{attribute 'qualified_only'}
{attribute 'strict'}
{attribute 'to_string'}
TYPE EOpenDichtSchuifStatus :
(
	Open := 0,
	Dicht,
	Error,
	Openen,
	Sluiten
);
END_TYPE

(* stored: Version 1.1.0.1
   DUT EOpenDichtSchuifStatus: Id {b27e2423-1a92-4315-b13f-123432824bdf} *)
